Yaskawa INFORM job: FRONT_WELD_90ST-1_5040.JBI

/JOB
//NAME FRONT_WELD_90ST-1_5040
///FOLDERNAME 02-SKRZYNIE_JOBS
//POS
///NPOS 28,28,0,6,0,0
///TOOL 0
///POSTYPE PULSE
///PULSE
C00000=0,-52278,40443,0,6873,1
C00001=0,-52278,40443,5610,-49281,72137
C00002=0,-42686,23640,7425,-34877,70985
C00003=25126,-44577,-4813,57071,-34461,49771
C00004=6017,-48449,-29001,102269,-8383,26407
C00005=2863,-32693,-8619,87056,-6043,33280
C00006=3232,-30428,-5975,86107,-6286,33771
C00007=-22659,-29440,-6589,78839,10459,34509
C00008=-48990,-22708,-2316,76239,27773,33219
C00009=-50847,-28145,-10545,73666,29314,34422
C00010=-71330,-4959,8771,57572,20266,52624
C00011=-72821,-3113,10678,58516,21171,52061
C00012=-72538,1249,18334,62867,20087,49895
C00013=-75784,1228,22240,77952,25383,45304
C00014=-69876,-3910,19536,86800,21295,42090
C00015=-54033,-13675,10685,97428,11103,38505
C00016=-58678,-17366,4552,88847,13968,42180
C00017=23545,-30165,-21390,32579,21562,60781
C00018=43411,-19640,-10965,-1347,18370,78573
C00019=44414,-17333,-7831,-3313,17976,79591
C00020=50382,-20084,-7461,-41259,20172,89579
C00021=52952,-20210,-9543,-47257,28986,86244
C00022=42056,-24733,-13162,-39378,23145,81494
C00023=22456,-29115,-21001,-6425,22404,64370
C00024=24971,-35737,-30976,-9397,24510,66000
C00025=0,-42686,23640,7425,-34877,70985
C00026=0,-52278,40443,5610,-49281,72137
C00027=0,-52278,40443,0,6873,1
BC00000=774759
BC00001=774759
BC00002=903040
BC00003=940675
BC00004=971500
BC00005=971500
BC00006=971501
BC00007=971502
BC00008=971501
BC00009=971501
BC00010=971502
BC00011=971502
BC00012=971502
BC00013=971502
BC00014=971562
BC00015=971502
BC00016=971502
BC00017=971502
BC00018=971501
BC00019=971501
BC00020=971501
BC00021=971501
BC00022=971501
BC00023=971501
BC00024=971501
BC00025=903040
BC00026=774759
BC00027=774759
///POSTYPE BASE
///RECTAN
///RCONF 1,0,0,0,0,0,0,0,0,0,0,0,0,0,0,0,0,0,0,0,0,0,0,0
P00500=2.332,-5.281,-1.258,0.0000,0.0000,0.0000
///RCONF 0,0,0,0,0,0,0,0,0,0,0,0,0,0,0,0,0,0,0,0,0,0,0,0
P00501=-2.026,0.009,3.534,0.0000,0.0000,0.0000
///RCONF 1,0,0,0,0,0,0,0,0,0,0,0,0,0,0,0,0,0,0,0,0,0,0,0
P00502=-2.023,0.001,1.732,0.0000,0.0000,0.0000
P00503=0.138,-0.044,1.539,0.0000,0.0000,0.0000
P00504=-0.309,-0.010,1.636,0.0000,0.0000,0.0000
P00505=0.999,-9.916,8.214,0.0000,0.0000,0.0000
//INST
///DATE 2024/05/13 20:09
///ATTR SC,RW
///GROUP1 RB1,BS1
NOP
MOVJ C00000 BC00000 VJ=50.00
MOVJ C00001 BC00001 VJ=50.00
MOVJ C00002 BC00002 VJ=50.00
MOVJ C00003 BC00003 VJ=50.00
MOVJ C00004 BC00004 VJ=30.00
'::::::::::::::::::::::::::::::::
'W20
'::::::::::::::::::::::::::::::::
MOVL C00005 BC00005 V=333.3
SFTON P0503
MACRO1 MJ#(0) ARGF14
MOVL C00006 BC00006 V=133.3 PL=0
ARCON
MOVL C00007 BC00007 V=9.5
SFTOF
SFTON P0502
MOVL C00008 BC00008 V=9.5
ARCOF
MOVL C00009 BC00009 V=250.0
SFTOF
MOVL C00010 BC00010 V=250.0
'::::::::::::::::::::::::::::::::
'W21
'::::::::::::::::::::::::::::::::
MOVL C00011 BC00011 V=166.7
SFTON P0500
MACRO1 MJ#(0) ARGF14
MOVL C00012 BC00012 V=133.3 PL=0
ARCON
MOVL C00013 BC00013 V=9.5
MOVL C00014 BC00014 V=9.5
SFTOF
SFTON P0501
MOVL C00015 BC00015 V=9.5
ARCOF
MOVL C00016 BC00016 V=250.0
SFTOF
MOVL C00017 BC00017 V=333.3
'::::::::::::::::::::::::::::::::
'W22
'::::::::::::::::::::::::::::::::
MOVL C00018 BC00018 V=166.7
SFTON P0505
MACRO1 MJ#(0) ARGF14
MOVL C00019 BC00019 V=133.3 PL=0
ARCON
MOVL C00020 BC00020 V=9.5
MOVL C00021 BC00021 V=9.5
SFTOF
SFTON P0504
MOVL C00022 BC00022 V=10.0
MOVL C00023 BC00023 V=10.0
ARCOF
MOVL C00024 BC00024 V=166.7
SFTOF
MOVJ C00025 BC00025 VJ=50.00
MOVJ C00026 BC00026 VJ=80.00
MOVJ C00027 BC00027 VJ=80.00
END
